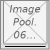
VISUALIZATION F_MainMenu_06  // 50x50
VAR_IN_OUT
	stMenuButton	: ST_HMIEButton_HMI;
END_VAR
    Image (3,0 44x44), image: ImagePool.06_Diagram
        OnMouseDown: execute { stMenuButton.bPushed := TRUE; }
    Line (5,46) (45,46), invisible if: not stMenuButton.bVisible or not stMenuButton.bActive, input disabled if: not stMenuButton.bEnable
END_VISUALIZATION

(* stored: Version 1.1.0.1
   Visu F_MainMenu_06: Id {cbf416d7-bca1-02b9-29de-865e7cac5c1f} *)
